// Mitsubishi GX Works2 project: 공압 프로젝트 1호기 2호기 2대운전 0924   PLC: Q03UDV

PROGRAM MAIN
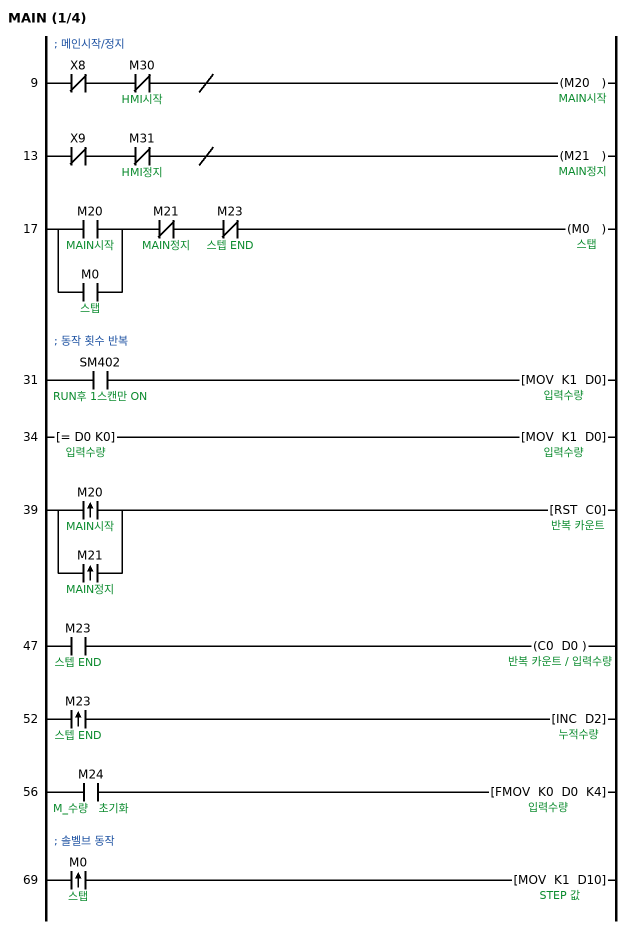
; 메인시작/정지
9     LDI     X8
      ANI     M30  ; HMI시작
      INV
      OUT     M20  ; MAIN시작
13    LDI     X9
      ANI     M31  ; HMI정지
      INV
      OUT     M21  ; MAIN정지
17    LD      M20  ; MAIN시작
      OR      M0  ; 스탭
      ANI     M21  ; MAIN정지
      ANI     M23  ; 스텝 END
      OUT     M0  ; 스탭
; 동작 횟수 반복
31    LD      SM402  ; RUN후 1스캔만 ON
      MOV     K1 D0  ; 입력수량
34    LD=     D0 K0  ; 입력수량
      MOV     K1 D0
39    LDP     M20  ; MAIN시작
      ORP     M21  ; MAIN정지
      RST     C0  ; 반복 카운트
47    LD      M23  ; 스텝 END
      OUT     C0 D0  ; 반복 카운트 / 입력수량
52    LDP     M23  ; 스텝 END
      INC     D2  ; 누적수량
56    LD      M24  ; M_수량   초기화
      FMOV    K0 D0 K4
; 솔벨브 동작
69    LDP     M0  ; 스탭
      MOV     K1 D10  ; STEP 값
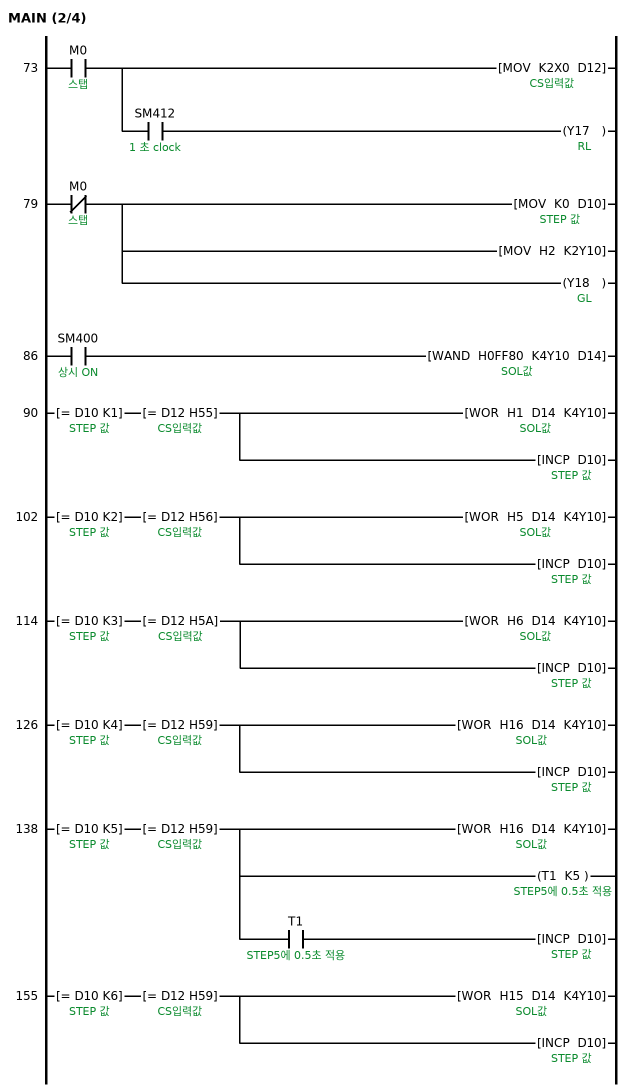
73    LD      M0  ; 스탭
      MOV     K2X0 D12  ; CS1        (후진) / CS입력값
      AND     SM412  ; 1 초 clock
      OUT     Y17  ; RL
79    LDI     M0  ; 스탭
      MOV     K0 D10
      MOV     H2 K2Y10  ; 양솔전진
      OUT     Y18  ; GL
86    LD      SM400  ; 상시 ON
      WAND    H0FF80 K4Y10 D14  ; SOL값
90    LD=     D10 K1  ; STEP 값
      AND=    D12 H55  ; CS입력값
      WOR     H1 D14 K4Y10
      INCP    D10
102   LD=     D10 K2  ; STEP 값
      AND=    D12 H56  ; CS입력값
      WOR     H5 D14 K4Y10
      INCP    D10
114   LD=     D10 K3  ; STEP 값
      AND=    D12 H5A  ; CS입력값
      WOR     H6 D14 K4Y10
      INCP    D10
126   LD=     D10 K4  ; STEP 값
      AND=    D12 H59  ; CS입력값
      WOR     H16 D14 K4Y10
      INCP    D10
138   LD=     D10 K5  ; STEP 값
      AND=    D12 H59  ; CS입력값
      WOR     H16 D14 K4Y10
      OUT     T1 K5  ; STEP5에 0.5초 적용
      AND     T1  ; STEP5에 0.5초 적용
      INCP    D10
155   LD=     D10 K6  ; STEP 값
      AND=    D12 H59  ; CS입력값
      WOR     H15 D14 K4Y10
      INCP    D10
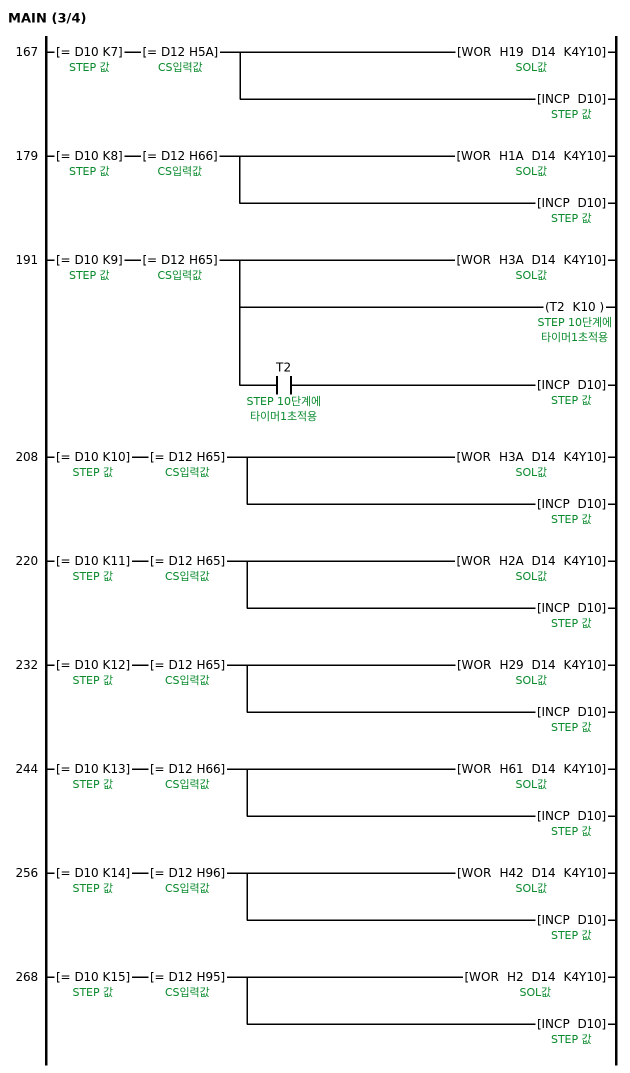
167   LD=     D10 K7  ; STEP 값
      AND=    D12 H5A  ; CS입력값
      WOR     H19 D14 K4Y10
      INCP    D10
179   LD=     D10 K8  ; STEP 값
      AND=    D12 H66  ; CS입력값
      WOR     H1A D14 K4Y10
      INCP    D10
191   LD=     D10 K9  ; STEP 값
      AND=    D12 H65  ; CS입력값
      WOR     H3A D14 K4Y10
      OUT     T2 K10  ; STEP 10단계에 타이머1초적용
      AND     T2  ; STEP 10단계에 타이머1초적용
      INCP    D10
208   LD=     D10 K10  ; STEP 값
      AND=    D12 H65  ; CS입력값
      WOR     H3A D14 K4Y10
      INCP    D10
220   LD=     D10 K11  ; STEP 값
      AND=    D12 H65  ; CS입력값
      WOR     H2A D14 K4Y10
      INCP    D10
232   LD=     D10 K12  ; STEP 값
      AND=    D12 H65  ; CS입력값
      WOR     H29 D14 K4Y10
      INCP    D10
244   LD=     D10 K13  ; STEP 값
      AND=    D12 H66  ; CS입력값
      WOR     H61 D14 K4Y10
      INCP    D10
256   LD=     D10 K14  ; STEP 값
      AND=    D12 H96  ; CS입력값
      WOR     H42 D14 K4Y10
      INCP    D10
268   LD=     D10 K15  ; STEP 값
      AND=    D12 H95  ; CS입력값
      WOR     H2 D14 K4Y10
      INCP    D10
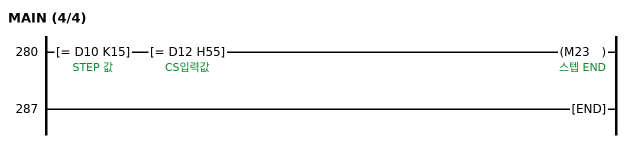
280   LD=     D10 K15  ; STEP 값
      AND=    D12 H55  ; CS입력값
      OUT     M23  ; 스텝 END
287   END
END_PROGRAM

// device comments not shown above
X1  ; CS2        (전진)
X2  ; CS3        (후진)
X3  ; CS4        (전진)
X4  ; 시작
X5  ; 정지
Y11  ; 양솔후진
Y12  ; 편솔
Y13  ; 부저
M1  ; 스탭 1
M2  ; 스탭 2
M3  ; 스탭 3
M4  ; 스텝 4
M5  ; 스텝5
M6  ; 스텝6
M7  ; 스텝7
M22  ; m 호밍(원상태 복귀)
M25  ; HMI 호밍
M32  ; RL
M33  ; YL
M34  ; GL
D11  ; 편솔
D20  ; CS_Step 번호
D22  ; CS_Val
D24  ; Sol_Val
T0  ; 타이머
